{attribute 'qualified_only'}
{attribute 'strict'}
TYPE eCyclinderTests : (
    Invalid := 25,
    StopMovement := 50,
    MoveHomeMoving := 100,
    MoveHomeMovingReached := 200,
    MoveWorkMoving := 300,
    MoveWorkMovingReached := 400,
    AbortMoveTask := 500,
    DisableHome := 600,
    DisableWork := 700,
    SuspendHome := 610,
    SuspendWork := 710,
    SuspendHomeInverted := 620,
    SuspendWorkInverted := 720,
    SuspendHomeExpression := 630,
    SuspendWorkExpression := 730
);
END_TYPE

(* stored: Version 1.1.0.1, ProductVersion 3.1.4024.12
   DUT eCyclinderTests: Id {32571aaf-264b-0000-0e82-067ca83bf104} *)
